FUNCTION_BLOCK Execute_State  IMPLEMENTS ITF_State
VAR_INPUT
END_VAR
VAR_OUTPUT
END_VAR
VAR
	pPML_Base : POINTER TO PML_StatePattern_Base;
	_stateMachine : IPmlStateMachine;
END_VAR

METHOD Cycle : BOOL
VAR_INPUT
END_VAR
IF _stateMachine.GetCurrentState() = E_PMLState.ePMLState_Aborting THEN
	pPML_Base^.SetState(pPML_Base^.aborting);
END_IF
END_METHOD

METHOD FB_init : BOOL
VAR_INPUT
	bInitRetains : BOOL; // if TRUE, the retain variables are initialized (warm start / cold start)
	bInCopyCode : BOOL;  // if TRUE, the instance afterwards gets moved into the copy code (online change)
	pPML_Base : POINTER TO PML_StatePattern_Base;
	statemachine : IPmlStateMachine;
END_VAR
_stateMachine := statemachine;
THIS^.pPML_Base := pPML_Base;
END_METHOD

END_FUNCTION_BLOCK

(* stored: Version 1.1.0.1, ProductVersion 3.1.4024.11
   POU Execute_State: Id {108202e6-c7c9-4974-a5b7-3acd91d8837a}, SpecialFunc None
   Method Cycle: Id {b81053a7-c788-40eb-a81c-996fff9d6b18}
   Method FB_init: Id {154cef4d-188f-4dcf-a46b-37b6c09094d7} *)
